// TIA Portal project "Project4" (V16)

(* hardware
DEVICE "S7-1200 station_1"  S7-1200 Station
   slot 0: "Rack_0"  S7-1200 Rack  Rack  V1.0
   slot 1: "PLC_1"  CPU 1214C DC/DC/DC  6ES7 214-1AG40-0XB0  V4.1
   slot 2: "DQ 16xRelay_1"  SM 1222 DQ16 x relay  6ES7 222-1HH32-0XB0  V2.0
   slot 3: "AQ 1x12BIT_1"  AQ1 signal board  6ES7 232-4HA30-0XB0  V1.0
*)

// ===== PLC "PLC_1"  CPU 1214C DC/DC/DC =====

VAR_GLOBAL   // PLC tag table "Default tag table"
   "Tag_1" AT %I0.2 : Bool;
   "Tag_2" AT %I0.1 : Bool;
   "Tag_3" AT %M0.0 : Bool;
   "Tag_4" AT %M0.5 : Bool;
   "Tag_5" AT %M1.2 : Bool;
   "Tag_6" AT %M0.4 : Bool;
   "Tag_7" AT %M0.1 : Bool;
   "Tag_8" AT %I0.3 : Bool;
   "Tag_9" AT %M0.3 : Bool;
   "Tag_10" AT %I0.7 : Bool;
   "Tag_11" AT %M1.1 : Bool;
   "Tag_12" AT %M1.3 : Bool;
   "Tag_13" AT %I0.4 : Bool;
   "Tag_14" AT %Q9.2 : Bool;
   "Tag_15" AT %Q9.3 : Bool;
   "Tag_16" AT %Q9.4 : Bool;
   "Tag_17" AT %Q9.5 : Bool;
   "Tag_18" AT %Q9.6 : Bool;
END_VAR

// folder: System blocks/Program resources

DATA_BLOCK "T1"   // DB1
{ S7_Optimized_Access := 'TRUE' }
AUTHOR : Simatic
FAMILY : IEC
NAME : IEC_TMR
VERSION : 1.0
// stored: InstanceOfName IEC_TIMER
"IEC_TIMER"
BEGIN
END_DATA_BLOCK

DATA_BLOCK "T2"   // DB2
{ S7_Optimized_Access := 'TRUE' }
AUTHOR : Simatic
FAMILY : IEC
NAME : IEC_TMR
VERSION : 1.0
// stored: InstanceOfName IEC_TIMER
"IEC_TIMER"
BEGIN
END_DATA_BLOCK

// folder: (top level)

ORGANIZATION_BLOCK "Main"   // OB1, LAD, ProgramCycle
TITLE = "Main Program Sweep (Cycle)"
{ S7_Optimized_Access := 'TRUE' }
VERSION : 0.1
   VAR_INPUT
      Initial_Call : Bool;   // Initial call of this OB
      Remanence : Bool;   // =True, if remanent data are available
   END_VAR
   VAR_TEMP   // added for the SCL form of the ladder/FBD networks
      _w1 : Bool;
   END_VAR
BEGIN

REGION Network 1
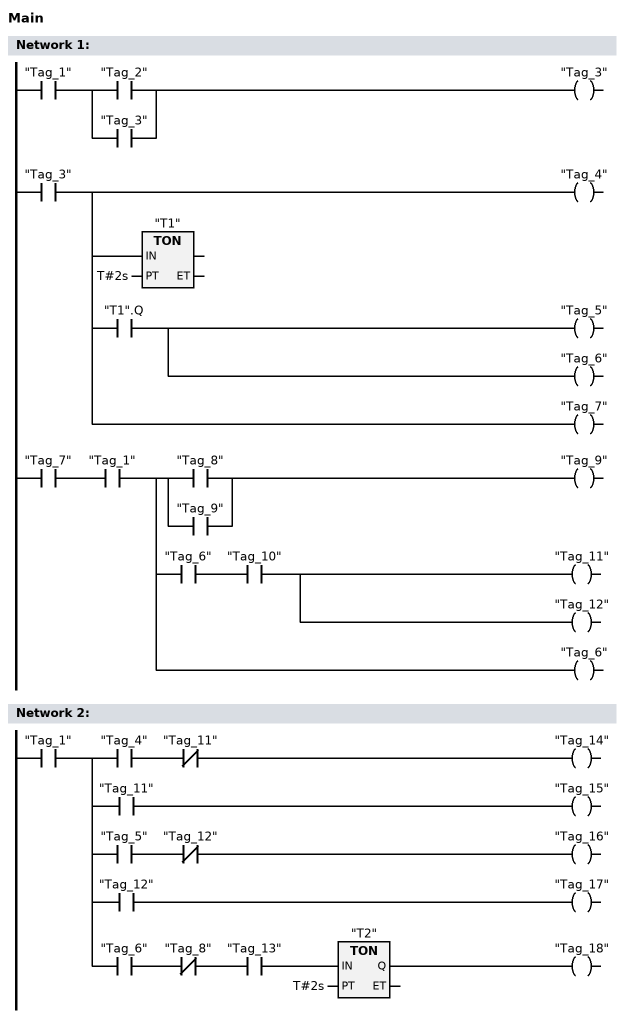
   "Tag_3" := "Tag_1" AND ("Tag_2" OR "Tag_3");
   "Tag_4" := "Tag_3";
   "T1".TON(IN := "Tag_3", PT := T#2s);
   "Tag_5" := "Tag_3" AND "T1".Q;
   "Tag_6" := "Tag_5";
   "Tag_7" := "Tag_3";
   #_w1 := "Tag_7" AND "Tag_1";
   "Tag_9" := #_w1 AND ("Tag_8" OR "Tag_9");
   "Tag_11" := #_w1 AND "Tag_6" AND "Tag_10";
   "Tag_12" := "Tag_11";
   "Tag_6" := #_w1;
END_REGION

REGION Network 2
   "Tag_14" := "Tag_1" AND "Tag_4" AND NOT "Tag_11";
   "Tag_15" := "Tag_1" AND "Tag_11";
   "Tag_16" := "Tag_1" AND "Tag_5" AND NOT "Tag_12";
   "Tag_17" := "Tag_1" AND "Tag_12";
   "T2".TON(IN := "Tag_1" AND "Tag_6" AND NOT "Tag_8" AND "Tag_13", PT := T#2s);
   "Tag_18" := "T2".Q;
END_REGION
END_ORGANIZATION_BLOCK